// TIA Portal V18 export
DATA_BLOCK "DB_FB_Robot_0"   // DB13
VERSION : 0.1
// stored: AutoNumber true, DBAccessibleFromOPCUA true, DBAccessibleFromWebserver true, InstanceOfName FB_Robot, InstanceOfType FB
"FB_Robot"
   // VAR_INPUT
   //    in_waypoint : Int;
   //    in_speed : Int;
   // END_VAR
   // VAR_OUTPUT
   //    out_succes : Bool;
   // END_VAR
   // VAR
   //    waypoints : Array[0..15] of "udt_Waypoint";
   // END_VAR
BEGIN
   // waypoints[2] : Caja Mediana in
   // waypoints[4] : Caja Mediana out
   // waypoints[5] : Caja Grande in
   // waypoints[6] : Caja Grande out
   // waypoints[7] : Caja Pequeña in
   // waypoints[8] : Caja Pequeña out
   waypoints[0..2].baseAxis := 90.0;
   waypoints[3..4].baseAxis := -93.0;
   waypoints[5].baseAxis := 90.0;
   waypoints[6].baseAxis := -93.0;
   waypoints[7].baseAxis := 90.0;
   waypoints[8].baseAxis := -93.0;
   waypoints[2].arm1Axis := 13.0;
   waypoints[3].arm1Axis := 0.0;
   waypoints[4].arm1Axis := 18.0;
   waypoints[5].arm1Axis := 13.0;
   waypoints[6].arm1Axis := 18.0;
   waypoints[7].arm1Axis := 16.0;
   waypoints[8].arm1Axis := 20.0;
   waypoints[2].arm2Axis := 18.0;
   waypoints[3].arm2Axis := 0.0;
   waypoints[4].arm2Axis := 6.0;
   waypoints[5].arm2Axis := 14.0;
   waypoints[6].arm2Axis := 0.0;
   waypoints[7].arm2Axis := 20.0;
   waypoints[8].arm2Axis := 10.0;
   waypoints[1].arm3Axis := 80.0;
   waypoints[2].arm3Axis := 58.0;
   waypoints[3].arm3Axis := 80.0;
   waypoints[4].arm3Axis := 64.0;
   waypoints[5].arm3Axis := 60.0;
   waypoints[6].arm3Axis := 68.0;
   waypoints[7].arm3Axis := 50.0;
   waypoints[8].arm3Axis := 58.0;
   waypoints[3..8].toolAxis := 0.0;
END_DATA_BLOCK
